PROGRAM MAIN
VAR
    fbLogHandler : FB_LogHandler;
END_VAR

fbLogHandler();

PRG_ECAT_CHECK();

PRG_GAUGES();

PRG_VALVES();

PRG_TURBO_PUMPS();

END_PROGRAM

(* stored: Version 1.1.0.1, ProductVersion 3.1.4024.12
   POU MAIN: Id {b66c7c96-5039-4af5-8cda-935a9b086c6f}, SpecialFunc None *)
